(* IEC 61131-3 sources: CodesysTest/export/Function Blocks/FB_Delay.pou, 1 file *)

(* ---- FB_Delay.pou.st ---- *)
(*#-#-#-#-#-#-#-#-#-#---Declaration---#-#-#-#-#-#-#-#-#-#-#-#-#*)

FUNCTION_BLOCK FB_Delay IMPLEMENTS IExecuteAutomatically
VAR_INPUT
	in : BOOL;
	delay : TIME;
END_VAR
VAR_OUTPUT
	Q : BOOL;
END_VAR
VAR
	delayTimer : TON;
END_VAR
(*#-#-#-#-#-#-#-#-#-#---Implementation---#-#-#-#-#-#-#-#-#-#-#-#-#*)
